FUNCTION_BLOCK TurnTableController
  (* Standard: 61499-2 *)
  (* Version 0.3, 2009-09-15, JHC, Holobloc Inc, Changed transition priorities. *)
  (* Version 0.2, 2003-12-04, JHC, Rockwell Automation, Renamed for better indexing. *)
  (* Version 0.1, 2002-11-05, JHC, Rockwell Automation, Corrected missing ST element in Algorithm REQ. *)
  (* Version 0.0, 2000-05-30, JHC, Rockwell Automation *)
  (* Compiler header: package fb.rt.dasdA1.A2.TurnTable; *)
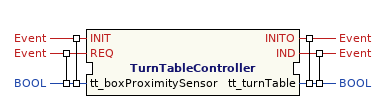
  EVENT_INPUT
    INIT WITH tt_boxProximitySensor; (* Initialization Request *)
    REQ WITH tt_boxProximitySensor;
  END_EVENT
  EVENT_OUTPUT
    INITO WITH tt_turnTable; (* Initialization Confirm *)
    IND WITH tt_turnTable; (* Execution Confirmation *)
  END_EVENT
  VAR_INPUT
    tt_boxProximitySensor : BOOL;
  END_VAR
  VAR_OUTPUT
    tt_turnTable : BOOL;
  END_VAR
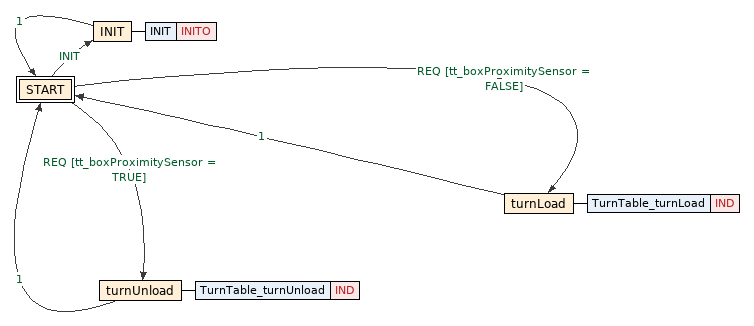
  EC_STATES
    START; (* Initial State *)
    INIT : INIT -> INITO; (* Initialization *)
    turnLoad : TurnTable_turnLoad -> IND;
    turnUnload : TurnTable_turnUnload -> IND;
  END_STATES
  EC_TRANSITIONS
    INIT TO START := 1;
    START TO INIT := INIT;
    START TO turnLoad := REQ [tt_boxProximitySensor = FALSE];
    turnLoad TO START := 1;
    START TO turnUnload := REQ [tt_boxProximitySensor = TRUE];
    turnUnload TO START := 1;
  END_TRANSITIONS
  ALGORITHM INIT IN ST: (* Initialization algorithm *)
tt_turnTable := FALSE;
  END_ALGORITHM
  ALGORITHM TurnTable_turnLoad IN ST:
tt_turnTable := FALSE;
  END_ALGORITHM
  ALGORITHM TurnTable_turnUnload IN ST:
tt_turnTable := TRUE;
  END_ALGORITHM
END_FUNCTION_BLOCK
